// TIA Portal V18 export
DATA_BLOCK "Speed_Control_SLS_DB"   // DB22, F_DB
// stored: InstanceOfName 01_Speed_Control_SLS, InstanceOfType FB
"01_Speed_Control_SLS"
   // VAR_INPUT
   //    PH1 : Bool;
   //    PH2 : Bool;
   //    SORTER_RUNNING_MSC : Bool;
   //    SLS_NOT_EN : Bool;
   //    RESET { ExternalWritable := 'False'} : Bool;
   //    "MIN[time]" : Time;
   //    "MAX[time]" : Time;
   //    "DelayRunning[time]" : Time;
   // END_VAR
   // VAR_OUTPUT
   //    SPEED_ZERO : Bool;
   //    SPEED_TOOHIGH : Bool;
   //    "PH1 Broken" : Bool;
   //    "PH2 Broken" : Bool;
   //    ENC_BROKEN : Bool;
   // END_VAR
   // VAR
   //    SR_RESET { ExternalWritable := 'False'} : Bool;
   //    Time_Limit : Time;
   //    TON_SLS_T_PH1 : TON;
   //    TON_SLS_T_PH2 : TON;
   //    TOF_PH1_WORKING : TOF;
   //    TOF_PH2_WORKING : TOF;
   //    TON_SORTER_STOP : TON;
   //    TON_TIMEOUT_COUNT : TON;
   //    TON_DELAY_RUNNING_STATUS : TON;
   //    CTU_SLS_PH1 : CTU;
   //    CTU_SLS_PH2 : CTU;
   //    PH1_FE : Bool;
   //    PH1_RE : Bool;
   //    PH2_FE : Bool;
   //    PH2_RE : Bool;
   //    PH1_ET : Time;
   //    PH2_ET : Time;
   //    BROKEN_FE : Bool;
   // END_VAR
BEGIN
END_DATA_BLOCK
